TYPE MyStruct :
STRUCT
sFilePath : STRING(1024);
sFolderPath : STRING(1024);

bTriggerNewFileSelected : BOOL;
bTriggerNewFolderSelected : BOOL;
END_STRUCT
END_TYPE

(* stored: Version 1.1.0.1, ProductVersion 3.1.4024.4
   DUT MyStruct: Id {d8d6d5d1-2aa6-4cd5-bf5f-31a38b8b06ba} *)
